// TIA Portal V19 export
DATA_BLOCK "ScreenNo"   // DB1
{ S7_Optimized_Access := 'TRUE' }
AUTHOR : FLA
FAMILY : UHT
VERSION : 1.0
// stored: AutoNumber false, MemoryReserve 0
   VAR RETAIN
      DW0 : Int;
      DW2 : Int;
      DW4 : Int;
      DW6 : Int;
      DW8 : Int;
      DW10 : Int;
      DW12 : Int;
   END_VAR
BEGIN
END_DATA_BLOCK
